// TIA Portal project "风机燃气" (V17)

(* hardware
DEVICE "PLC_1"  S7-1200 Station
   slot 0: "Rack_0"  S7-1200 Rack  Rack  V1.0
   slot 1: "PLC_1"  CPU 1214C DC/DC/DC  6ES7 214-1AG40-0XB0  V4.5
*)

// ===== PLC "PLC_1"  CPU 1214C DC/DC/DC =====

VAR_GLOBAL   // PLC tag table "IO变量"
   "风机运行" AT %Q4.4 : Bool;
   "烧嘴电源" AT %Q4.6 : Bool;
   "风机控制" AT %QW44 : Word;
END_VAR

DATA_BLOCK "信号数据"   // DB1
{ S7_Optimized_Access := 'TRUE' }
VERSION : 0.1
   VAR
      风机运行按 : Bool;
      风机故障反馈 : Bool;
      风机手动 : Bool;
      风机自动输出 : Real;
      风机手动频率 : Real;
      风机控制输出 : Real;
      风压测量值 : Real;
   END_VAR
BEGIN
END_DATA_BLOCK

FUNCTION "FC_风机燃气控制" : Void   // FC1, LAD
{ S7_Optimized_Access := 'TRUE' }
   VAR_TEMP
      风机控制输出值 : Real;
      风压过渡 : Int;
   END_VAR
BEGIN

REGION Network 1: 风机运行控制
   // 常开触点风机运行按与常闭触点风机故障反馈串联，当风机运行按接通且风机故障反馈未动作时，驱动风机运行线圈Q4.4
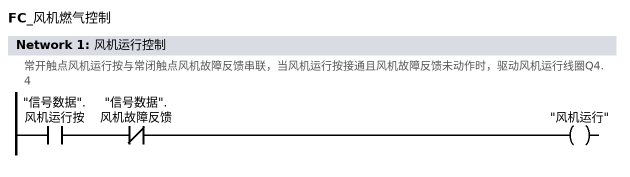
   RUNG wire#powerrail
      Contact( "信号数据".风机运行按 )
      I_Contact( "信号数据".风机故障反馈 )
      Coil( "风机运行" )
   END_RUNG
   // the same network as SCL:
   "风机运行" := "信号数据".风机运行按 AND NOT "信号数据".风机故障反馈;
END_REGION
END_FUNCTION

ORGANIZATION_BLOCK "Main"   // OB1, LAD, ProgramCycle
TITLE = "Main Program Sweep (Cycle)"
{ S7_Optimized_Access := 'TRUE' }
VERSION : 0.1
   VAR_INPUT
      Initial_Call : Bool;   // Initial call of this OB
      Remanence : Bool;   // =True, if remanent data are available
   END_VAR
BEGIN
END_ORGANIZATION_BLOCK